(* PLC project Unnamed, Unknown Unnamed 1 *)
(* stored: creationDateTime 2026-02-02T16:17:06, modificationDateTime 2026-02-02T16:17:06 *)

PROGRAM main
  VAR
    LocalVar : DINT;
  END_VAR

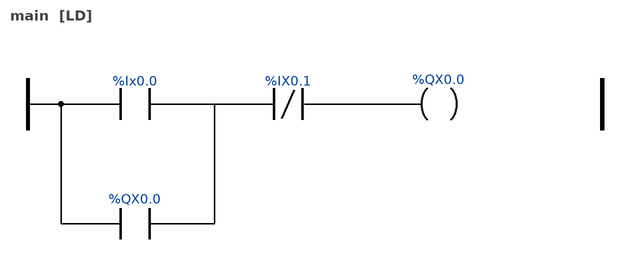
(* LD diagram, written out as Structured Text *)
%QX0.0 := (%Ix0.0 OR %QX0.0) AND NOT %IX0.1;
END_PROGRAM

CONFIGURATION Config0
  RESOURCE Res0 ON PLC
    TASK task0(INTERVAL := T#20ms, PRIORITY := 1);
    PROGRAM instance0 WITH task0 : main;
  END_RESOURCE
END_CONFIGURATION
